(* CODESYS project emBRICK_demo.project

Project tree, tasks and I/O mapping:
  Device : CODESYS Control Win V3, 3S - Smart Software Solutions GmbH, version 3.5.16.40
    application Application
      libraries: Standard, * (System)
      task MainTask (cyclic, interval t#10ms, priority 1) calls POU
      task VISU_TASK (cyclic, interval 100 ms, priority 31) calls VisuElems.Visu_Prg
      program POU [ST]
      data type STATE
      visualisation Visualization
      program POU_ohneMapping [ST]
    CAE_Z_PadBridgeMX : CAE_Z-PatBridgeMX, emBRICK GmbH, order no. VIM0-0204A00, version 1.6
        settings: COM Port = 5
      CAE_P_2Rel4Di2Ai_01 : CAE_P-2Rel4Di2Ai-01, emBRICK GmbH, order no. VIM0-0150A00, version 1.0
          input  Application.POU.ai_2Rel4Di2Ai[0] :  WORD  // Analog Input 1
          input  Application.POU.ai_2Rel4Di2Ai[1] :  WORD  // Analog Input 2
          input  Application.POU.di_2Rel4Di2Ai[0] : BOOL  // Digital Input.Bit0
          input  Application.POU.di_2Rel4Di2Ai[1] : BOOL  // Digital Input.Bit1
          input  Application.POU.di_2Rel4Di2Ai[2] : BOOL  // Digital Input.Bit2
          input  Application.POU.di_2Rel4Di2Ai[3] : BOOL  // Digital Input.Bit3
          output Application.POU.relais_2Rel4Di2Ai[0] : BOOL  // Relays.Bit0
          output Application.POU.relais_2Rel4Di2Ai[1] : BOOL  // Relays.Bit1
          unmapped channels: Status, Digital Input, Relays
  libraries: VisuSymbols, 3.5.10.0 (System)
  text list GlobalTextList
*)

// Device/Application/STATE
TYPE STATE :
(
	INIT := 0,
	RUNNING := 1
);
END_TYPE

// Device/Application/POU
PROGRAM POU
VAR_INPUT
	// Settings
	callTimeMS : UINT := 10;	// Cycle Time in [ms]	

	// I/Os
	relais_2Rel4Di2Ai : ARRAY[0..1] OF BOOL;
	di_2Rel4Di2Ai : ARRAY[0..3] OF BOOL;
	ai_2Rel4Di2Ai : ARRAY[0..1] OF WORD;
	
	// Helpers
	taskCounter : DWORD := 0;
	oldTaskCounter : DWORD := 0;
END_VAR

taskCounter := taskCounter + 1;
(* - IOs should be updated atleast once every 100ms *)	

// Example Application
	
// Toggle Relais 1 every Second
IF ((taskCounter - oldTaskCounter) * callTimeMS) > 1000 THEN
	IF relais_2Rel4Di2Ai[0] = TRUE THEN
		relais_2Rel4Di2Ai[0] := FALSE;
	ELSE
		relais_2Rel4Di2Ai[0] := TRUE;
	END_IF
	oldTaskCounter := taskCounter;
END_IF

// Switch Relais 2 to Value on Input 1
relais_2Rel4Di2Ai[1] := di_2Rel4Di2Ai[0];

END_PROGRAM

// Device/Application/POU_ohneMapping
PROGRAM POU_ohneMapping
VAR
	// Settings
	callTimeMS : UINT := 10;	// Cycle Time in [ms]
	// Helpers
	taskCounter : DWORD := 0;
	oldTaskCounter : DWORD := 0;
END_VAR

taskCounter := taskCounter + 1;

(* - IOs should be updated once every 100ms *)	

// Example Application
// without Mapping you can Controll your IO's with the variable name and with her Adress
// Relais1 has the Adress %QX0.0
// Relais2 has the Adress %QX0.1
// Toggle Relais 1  every Second
IF ((taskCounter - oldTaskCounter) * callTimeMS) > 1000 THEN
	// Here we take the variable name
	IF Relais1 = TRUE THEN
		// But we can easily work with the adress to
		%QX0.0 := FALSE;
		// Relais1 = TRUE
	ELSE
		Relais1 := TRUE;
	END_IF
	oldTaskCounter := taskCounter;
END_IF

// Switch Relais 2 to Value on Input 1
%QX0.1 := DI1;
//Relais2 := DI1;

END_PROGRAM

// Device/Application/Visualization
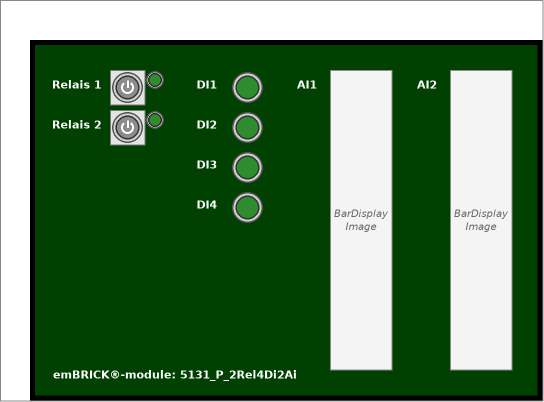
VISUALIZATION Visualization  // 544x402
    Rectangle (30,40 512x360)
    Lamp1 (230,70 35x35), variable: POU.di_2Rel4Di2Ai[0], style: Lamp-Lamp1-Green
    Lamp1 (145,70 20x20), variable: POU.relais_2Rel4Di2Ai[0], style: Lamp-Lamp1-Green
    PowerSwitch (110,70 35x35), variable: POU.relais_2Rel4Di2Ai[0], behaviour: TOGGLE, style: Switch-PowerSwitch-Gray
    Lamp1 (145,110 20x20), variable: POU.relais_2Rel4Di2Ai[1], style: Lamp-Lamp1-Green
    PowerSwitch (110,110 35x35), variable: POU.relais_2Rel4Di2Ai[1], behaviour: TOGGLE, style: Switch-PowerSwitch-Gray
    Lamp1 (230,110 35x35), variable: POU.di_2Rel4Di2Ai[1], style: Lamp-Lamp1-Green
    Lamp1 (230,150 35x35), variable: POU.di_2Rel4Di2Ai[2], style: Lamp-Lamp1-Green
    Lamp1 (230,190 35x35), variable: POU.di_2Rel4Di2Ai[3], style: Lamp-Lamp1-Green
    BarDisplayImage (450,70 62x300), value: POU.ai_2Rel4Di2Ai[1], style: BarDisplayImage-Gray, scale format: %.0f, scale 0..1100
    Label (50,70 54x30), "Relais 1"
    Label (50,110 54x30), "Relais 2"
    Label (180,70 54x30), "DI1"
    Label (180,110 54x30), "DI2"
    Label (180,150 54x30), "DI3"
    Label (180,190 54x30), "DI4"
    Label (280,70 54x30), "AI1"
    Label (400,70 54x30), "AI2"
    BarDisplayImage (330,70 62x300), value: POU.ai_2Rel4Di2Ai[0], style: BarDisplayImage-Gray, scale format: %.0f, scale 0..1100
    Label (50,360 238x30), "emBRICK®-module: 5131_P_2Rel4Di2Ai"
END_VISUALIZATION
